(* CoDeSys 2.3 export: TYPE_LED_RGB.EXP *)

(* Data type *)
TYPE Type_LED_RGB :
STRUCT
	Hue				:REAL;
	Saturation			:REAL:= 100.0;
	Brightness			:REAL:=100;
	Switch_ON			:BOOL;
	Switch_RANDOM	:BOOL;
	Config				:Type_LED_RGB_CONFIG;
	Red					:BYTE;
	Green				:BYTE;
	Blue				:BYTE;
END_STRUCT
END_TYPE
